// TwinCAT 3 PLC project calibrateio
// ProgramVersion: 3.1.0.8
// libraries:
//   Tc2_Standard, * (Beckhoff Automation GmbH)
//   Tc2_System, * (Beckhoff Automation GmbH)
//   Tc3_Interfaces, * (Beckhoff Automation GmbH)
//   Tc3_Module, * (Beckhoff Automation GmbH)
// project tree:
//   GVLs/ GVL.TcGVL
//   / PlcTask.TcTTO
//   POUs/ MAIN.TcPOU
// real-time tasks:
//   TASK PlcTask: cycle T#10ms, priority 20, ADS port 350
// I/O:
//   DEVICE Device 1 (EtherCAT), AmsNetId 5.20.215.224.2.1
//     Term 1 (EK1200) [EK1200-5000 EtherCAT Power supply (2A E-Bus)]
//       Term 2 (EL3058) [EL3058 8Ch. Ana. Input 4-20mA]
//       Term 3 (EL4028) [EL4028 8Ch. Ana. Output 4-20mA, 12bit]
//       Term 4 (EL1808) [EL1808 8Ch. Dig. Input 24V, 3ms]
//       Term 5 (EL2808) [EL2808 8Ch. Dig. Output 24V, 0.5A]
//       Term 6 (EL3068) [EL3068 8Ch. Ana. Input 0-10V]
//       Term 7 (EL4008) [EL4008 8Ch. Ana. Output 0-10V, 12bit]
//       Term 8 (EL9011) [EL9011 End Terminal]
// variable links:
//   calibrateio/calibrateio Instance <-> Device 1 (EtherCAT)/Term 1 (EK1200)/Term 2 (EL3058)
//     PlcTask Inputs/GVL.XIN[{1..8}] <-> AI Standard Channel {1..8}/Value  (8 links)
//   calibrateio/calibrateio Instance <-> Device 1 (EtherCAT)/Term 1 (EK1200)/Term 3 (EL4028)
//     PlcTask Outputs/GVL.XOUT[{1..8}] <-> AO Outputs Channel {1..8}/Analog output  (8 links)

CONFIGURATION calibrateio
    RESOURCE PLC ON TwinCAT3
        TASK PlcTask(INTERVAL := T#10ms, PRIORITY := 20);
        PROGRAM MAIN WITH PlcTask : MAIN;
    END_RESOURCE
END_CONFIGURATION

// ---- GVLs/GVL.TcGVL
VAR_GLOBAL
	
	// IO Calibration parameters
	NL:INT:=4000;
	NH:INT:=32000;
	NSTEP:INT:=4000;
	NRANGE: INT;
	
	// IO mapping
	NIO : INT := 8;
	XOUT AT %Q*	:	ARRAY[1..8] OF INT :=[8(0)];
	XIN	AT %I*	:	ARRAY[1..8] OF INT :=[8(0)];
	
	// calibration measurement
	DELTA	:	ARRAY[1..8, 1..8] OF LREAL := [8(0.0), 8(0.0)];
	
END_VAR

// ---- POUs/MAIN.TcPOU
PROGRAM MAIN
VAR
	
	GO	: BOOL	:=	FALSE;	

	pv	:	INT := 0;
	xhat : ARRAY[1..8] OF LREAL;
	xsum : ARRAY[1..8] OF LREAL;

	ii:INT:=0;
	jj:INT:=0;
	kk:LREAL:=1.0;
	
	Tset: TON := (IN := TRUE, PT := TIME#10S, Q:=TRUE);
	
END_VAR


NRANGE:=NH/NSTEP;
IF GO AND jj<=NRANGE THEN 
	
	Tset(IN:=NOT(Tset.Q));
	
	IF Tset.Q OR (jj=0) THEN 
		
		jj := jj + 1;
		pv := jj*NSTEP;
		
		FOR ii := 1 TO NIO DO	
			// set the output level
			XOUT[ii] := pv;
			// reset measurement counter
			xhat[ii] := 0.0;
			xsum[ii] := 0.0;		
		END_FOR
		
		kk := 1;
		
	END_IF
	
	// take the measurements
	IF kk > 300 THEN
		FOR ii := 1 TO NIO DO
			//xhat[ii] := alpha*XIN[ii] + (1-alpha)*xhat[ii];
			xsum[ii] := xsum[ii] + XIN[ii];
			xhat[ii] := xsum[ii]/(kk-300);
			DELTA[ii,jj] := INT_TO_LREAL(XOUT[ii]) - xhat[ii];
		END_FOR
	END_IF
	
	// increment meas counter each scan
	kk := kk + 1;

END_IF

END_PROGRAM
